(*

short summary
=============

.. <legal notes>

legal notes
=================
| SPDX-FileCopyrightText: © 2023 ekvip automation GmbH <info@ekvip.de>
| SPDX-License-Identifier: Apache-2.0
| For details check: Apache-2.0_

.. _Apache-2.0: https://www.apache.org/licenses/LICENSE-2.0

.. </legal notes>

enumeration values
==================

*)

{warning 'header is generated please add your documentation'}
{attribute 'qualified_only'}
{attribute 'strict'}
{attribute 'to_string'}
TYPE StringType :
(
	ASCII_STRING := 0,
	UTF16STRING  := 1
)USINT;
END_TYPE

(* stored: Version 1.1.0.1, ProductVersion 3.1.4024.12
   DUT StringType: Id {165f7093-2cd6-4c05-948d-43958bf40c7a} *)
